SYSTEM TRAFFIC_LIGHT_CENTRALIZED (* System Configuration *)
  (* Standard: 61499-1 *)
  (* Version 0.4, 2009-03-05, JHC, Holobloc Inc., Deleted Application. *)
  (* Version 0.3, 2003-12-05, JHC, Rockwell Automation, Renamed from NEWSYSTEM. *)
  (* Version 0.2, 2002-11-05, JHC, Rockwell Automation, Fixed missing (empty) FBD in Application. *)
  (* Version 0.1, 2002-01-17, JHC, Rockwell Automation, Minor cleanup *)
  (* Version 0.0, 2000-05-27, JHC, Rockwell Automation *)
  DEVICE HMI_ROAD3_ROAD4 : FRAME_DEVICE(GRID := [2,1], BOUNDS := [10,10,300,500])
    RESOURCE HMI_ROAD3 : PANEL_RESOURCE
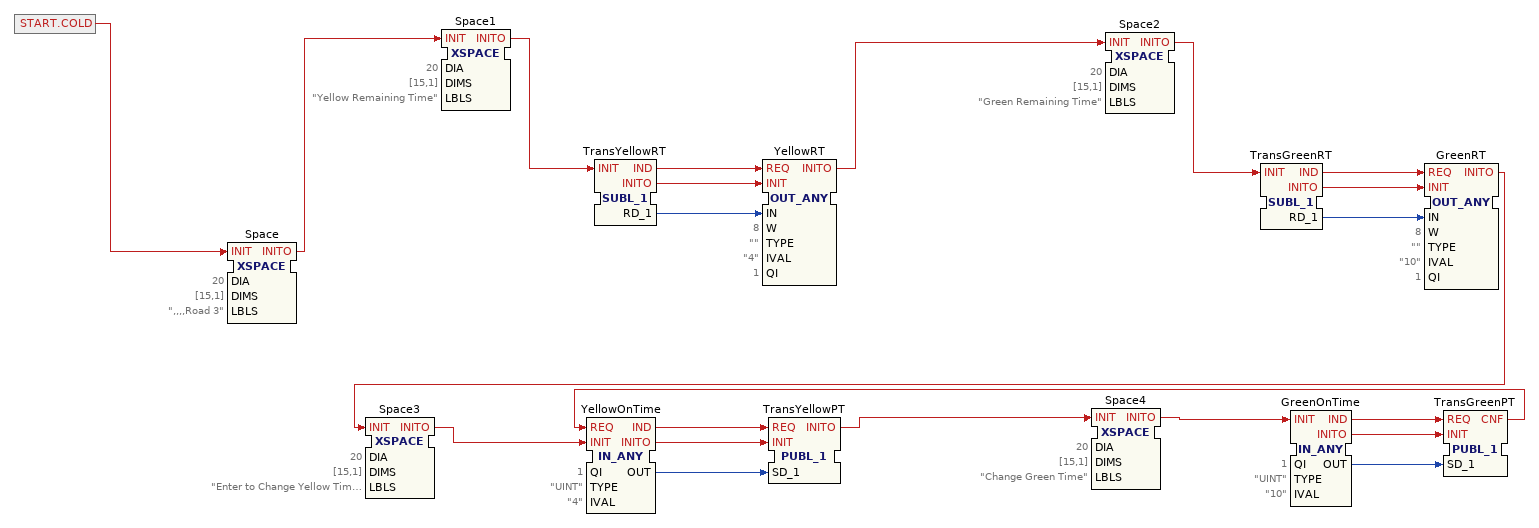
      FBS
        YellowRT : OUT_ANY(W := 8, TYPE := "", IVAL := "4", QI := 1);
        GreenRT : OUT_ANY(W := 8, TYPE := "", IVAL := "10", QI := 1);
        TransYellowRT : SUBL_1;
        TransGreenRT : SUBL_1;
        TransGreenPT : PUBL_1;
        TransYellowPT : PUBL_1;
        GreenOnTime : IN_ANY(QI := 1, TYPE := "UINT", IVAL := "10");
        YellowOnTime : IN_ANY(QI := 1, TYPE := "UINT", IVAL := "4");
        Space2 : XSPACE(DIA := 20, DIMS := [15,1], LBLS := "Green Remaining Time");
        Space1 : XSPACE(DIA := 20, DIMS := [15,1], LBLS := "Yellow Remaining Time");
        Space3 : XSPACE(DIA := 20, DIMS := [15,1], LBLS := "Enter to Change  Yellow Time");
        Space4 : XSPACE(DIA := 20, DIMS := [15,1], LBLS := "Change  Green Time");
        Space : XSPACE(DIA := 20, DIMS := [15,1], LBLS := ",,,,Road 3");
      END_FBS
      EVENT_CONNECTIONS
        TransYellowRT.IND TO YellowRT.REQ;
        TransGreenRT.IND TO GreenRT.REQ;
        YellowOnTime.IND TO TransYellowPT.REQ;
        GreenOnTime.IND TO TransGreenPT.REQ;
        YellowOnTime.INITO TO TransYellowPT.INIT;
        GreenOnTime.INITO TO TransGreenPT.INIT;
        TransGreenPT.CNF TO YellowOnTime.REQ;
        TransGreenRT.INITO TO GreenRT.INIT;
        YellowRT.INITO TO Space2.INIT;
        Space2.INITO TO TransGreenRT.INIT;
        TransYellowRT.INITO TO YellowRT.INIT;
        Space1.INITO TO TransYellowRT.INIT;
        GreenRT.INITO TO Space3.INIT;
        Space3.INITO TO YellowOnTime.INIT;
        TransYellowPT.INITO TO Space4.INIT;
        Space4.INITO TO GreenOnTime.INIT;
        START.COLD TO Space.INIT;
        Space.INITO TO Space1.INIT;
      END_CONNECTIONS
      DATA_CONNECTIONS
        TransYellowRT.RD_1 TO YellowRT.IN;
        TransGreenRT.RD_1 TO GreenRT.IN;
        YellowOnTime.OUT TO TransYellowPT.SD_1;
        GreenOnTime.OUT TO TransGreenPT.SD_1;
      END_CONNECTIONS
    END_RESOURCE
    RESOURCE HMI_ROAD4 : PANEL_RESOURCE
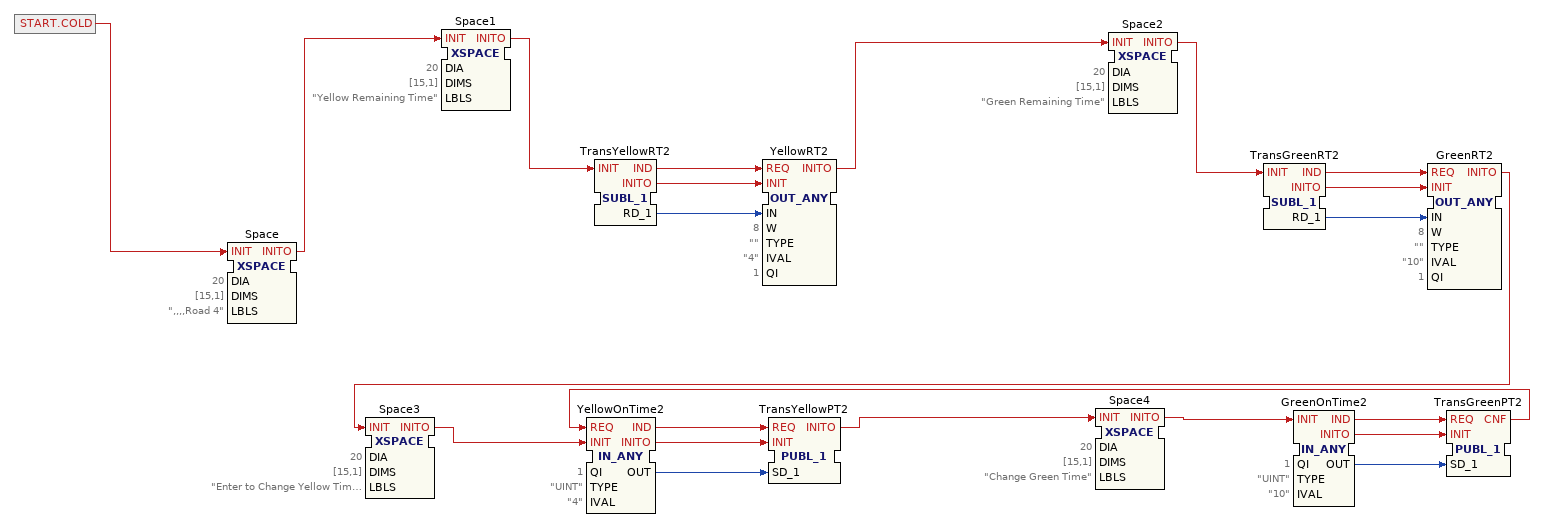
      FBS
        YellowRT2 : OUT_ANY(W := 8, TYPE := "", IVAL := "4", QI := 1);
        GreenRT2 : OUT_ANY(W := 8, TYPE := "", IVAL := "10", QI := 1);
        TransYellowRT2 : SUBL_1;
        TransGreenRT2 : SUBL_1;
        TransGreenPT2 : PUBL_1;
        TransYellowPT2 : PUBL_1;
        GreenOnTime2 : IN_ANY(QI := 1, TYPE := "UINT", IVAL := "10");
        YellowOnTime2 : IN_ANY(QI := 1, TYPE := "UINT", IVAL := "4");
        Space2 : XSPACE(DIA := 20, DIMS := [15,1], LBLS := "Green Remaining Time");
        Space1 : XSPACE(DIA := 20, DIMS := [15,1], LBLS := "Yellow Remaining Time");
        Space3 : XSPACE(DIA := 20, DIMS := [15,1], LBLS := "Enter to Change  Yellow Time");
        Space4 : XSPACE(DIA := 20, DIMS := [15,1], LBLS := "Change  Green Time");
        Space : XSPACE(DIA := 20, DIMS := [15,1], LBLS := ",,,,Road 4");
      END_FBS
      EVENT_CONNECTIONS
        TransYellowRT2.IND TO YellowRT2.REQ;
        TransGreenRT2.IND TO GreenRT2.REQ;
        YellowOnTime2.IND TO TransYellowPT2.REQ;
        GreenOnTime2.IND TO TransGreenPT2.REQ;
        YellowOnTime2.INITO TO TransYellowPT2.INIT;
        GreenOnTime2.INITO TO TransGreenPT2.INIT;
        TransGreenPT2.CNF TO YellowOnTime2.REQ;
        TransGreenRT2.INITO TO GreenRT2.INIT;
        YellowRT2.INITO TO Space2.INIT;
        Space2.INITO TO TransGreenRT2.INIT;
        TransYellowRT2.INITO TO YellowRT2.INIT;
        Space1.INITO TO TransYellowRT2.INIT;
        GreenRT2.INITO TO Space3.INIT;
        Space3.INITO TO YellowOnTime2.INIT;
        TransYellowPT2.INITO TO Space4.INIT;
        Space4.INITO TO GreenOnTime2.INIT;
        START.COLD TO Space.INIT;
        Space.INITO TO Space1.INIT;
      END_CONNECTIONS
      DATA_CONNECTIONS
        TransYellowRT2.RD_1 TO YellowRT2.IN;
        TransGreenRT2.RD_1 TO GreenRT2.IN;
        YellowOnTime2.OUT TO TransYellowPT2.SD_1;
        GreenOnTime2.OUT TO TransGreenPT2.SD_1;
      END_CONNECTIONS
    END_RESOURCE
  END_DEVICE
  DEVICE VIEW_ROAD3_ROAD4 : FRAME_DEVICE(BOUNDS := [310,10,300,500], GRID := [2,1])
    RESOURCE VIEW_ROAD3 : PANEL_RESOURCE(ROWS := 0, COLS := 0)
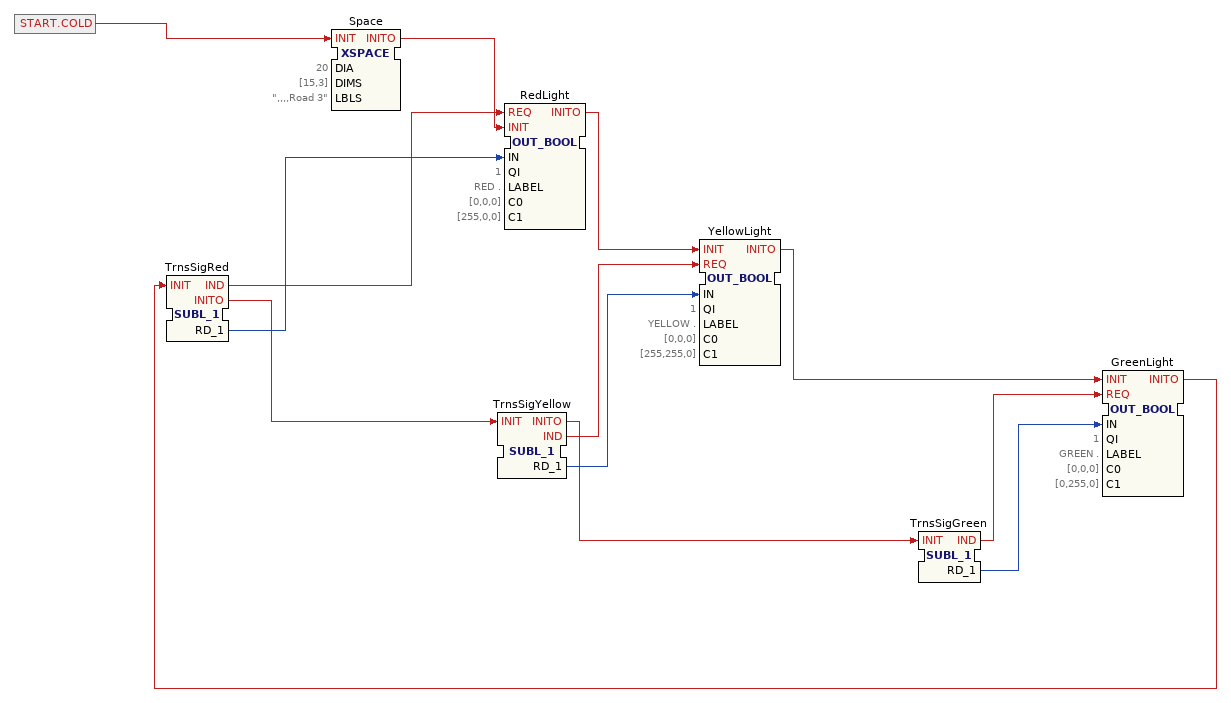
      FBS
        TrnsSigRed : SUBL_1;
        YellowLight : OUT_BOOL(QI := 1, LABEL := YELLOW    ., C0 := [0,0,0], C1 := [255,255,0]);
        RedLight : OUT_BOOL(QI := 1, LABEL := RED    ., C0 := [0,0,0], C1 := [255,0,0]);
        GreenLight : OUT_BOOL(QI := 1, LABEL := GREEN    ., C0 := [0,0,0], C1 := [0,255,0]);
        TrnsSigYellow : SUBL_1;
        TrnsSigGreen : SUBL_1;
        Space : XSPACE(DIA := 20, DIMS := [15,3], LBLS := ",,,,Road 3");
      END_FBS
      EVENT_CONNECTIONS
        RedLight.INITO TO YellowLight.INIT;
        YellowLight.INITO TO GreenLight.INIT;
        GreenLight.INITO TO TrnsSigRed.INIT;
        TrnsSigRed.IND TO RedLight.REQ;
        TrnsSigRed.INITO TO TrnsSigYellow.INIT;
        TrnsSigYellow.INITO TO TrnsSigGreen.INIT;
        TrnsSigYellow.IND TO YellowLight.REQ;
        TrnsSigGreen.IND TO GreenLight.REQ;
        START.COLD TO Space.INIT;
        Space.INITO TO RedLight.INIT;
      END_CONNECTIONS
      DATA_CONNECTIONS
        TrnsSigRed.RD_1 TO RedLight.IN;
        TrnsSigYellow.RD_1 TO YellowLight.IN;
        TrnsSigGreen.RD_1 TO GreenLight.IN;
      END_CONNECTIONS
    END_RESOURCE
    RESOURCE VIEW_ROAD4 : PANEL_RESOURCE(ROWS := 0, COLS := 0)
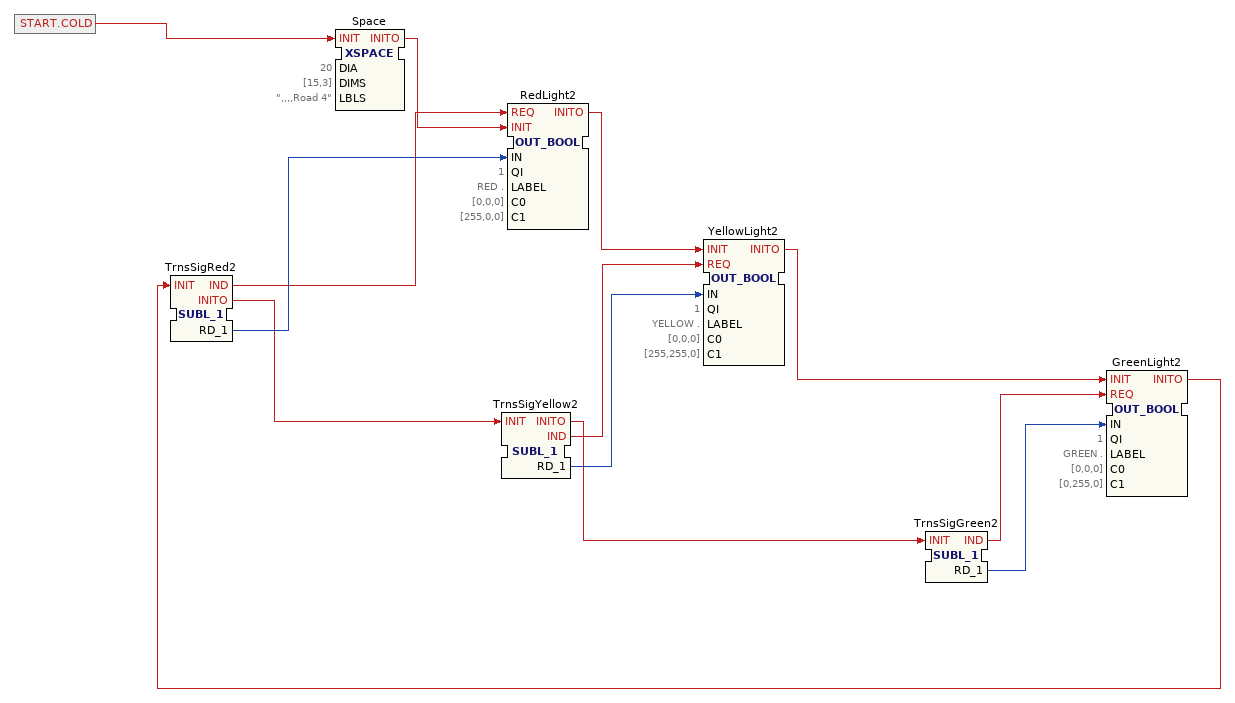
      FBS
        TrnsSigRed2 : SUBL_1;
        YellowLight2 : OUT_BOOL(QI := 1, LABEL := YELLOW    ., C0 := [0,0,0], C1 := [255,255,0]);
        RedLight2 : OUT_BOOL(QI := 1, LABEL := RED    ., C0 := [0,0,0], C1 := [255,0,0]);
        GreenLight2 : OUT_BOOL(QI := 1, LABEL := GREEN    ., C0 := [0,0,0], C1 := [0,255,0]);
        TrnsSigYellow2 : SUBL_1;
        TrnsSigGreen2 : SUBL_1;
        Space : XSPACE(DIA := 20, DIMS := [15,3], LBLS := ",,,,Road 4");
      END_FBS
      EVENT_CONNECTIONS
        RedLight2.INITO TO YellowLight2.INIT;
        YellowLight2.INITO TO GreenLight2.INIT;
        GreenLight2.INITO TO TrnsSigRed2.INIT;
        TrnsSigRed2.IND TO RedLight2.REQ;
        TrnsSigRed2.INITO TO TrnsSigYellow2.INIT;
        TrnsSigYellow2.INITO TO TrnsSigGreen2.INIT;
        TrnsSigYellow2.IND TO YellowLight2.REQ;
        TrnsSigGreen2.IND TO GreenLight2.REQ;
        START.COLD TO Space.INIT;
        Space.INITO TO RedLight2.INIT;
      END_CONNECTIONS
      DATA_CONNECTIONS
        TrnsSigRed2.RD_1 TO RedLight2.IN;
        TrnsSigYellow2.RD_1 TO YellowLight2.IN;
        TrnsSigGreen2.RD_1 TO GreenLight2.IN;
      END_CONNECTIONS
    END_RESOURCE
  END_DEVICE
  DEVICE MODEL_ROAD3_ROAD4 : FRAME_DEVICE(BOUNDS := [0,0,0,0], GRID := [1,1])
    RESOURCE MODEL_ROAD3 : PANEL_RESOURCE(ROWS := 0, COLS := 0)
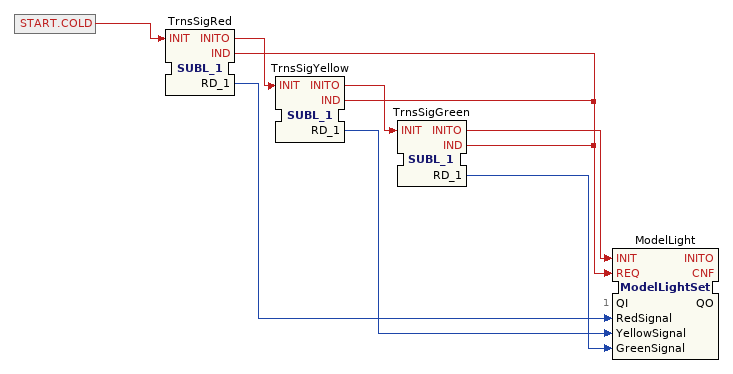
      FBS
        TrnsSigRed : SUBL_1;
        TrnsSigYellow : SUBL_1;
        TrnsSigGreen : SUBL_1;
        ModelLight : ModelLightSet(QI := 1);
      END_FBS
      EVENT_CONNECTIONS
        TrnsSigRed.INITO TO TrnsSigYellow.INIT;
        TrnsSigYellow.INITO TO TrnsSigGreen.INIT;
        START.COLD TO TrnsSigRed.INIT;
        TrnsSigGreen.INITO TO ModelLight.INIT;
        TrnsSigGreen.IND TO ModelLight.REQ;
        TrnsSigYellow.IND TO ModelLight.REQ;
        TrnsSigRed.IND TO ModelLight.REQ;
      END_CONNECTIONS
      DATA_CONNECTIONS
        TrnsSigRed.RD_1 TO ModelLight.RedSignal;
        TrnsSigYellow.RD_1 TO ModelLight.YellowSignal;
        TrnsSigGreen.RD_1 TO ModelLight.GreenSignal;
      END_CONNECTIONS
    END_RESOURCE
    RESOURCE MODEL_ROAD4 : PANEL_RESOURCE(ROWS := 0, COLS := 0)
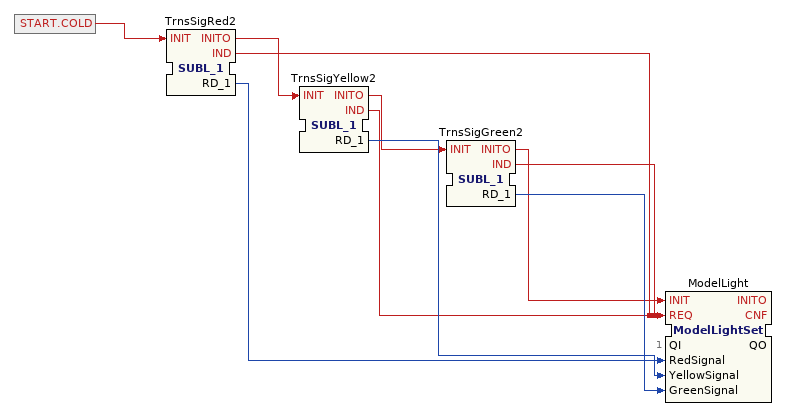
      FBS
        TrnsSigRed2 : SUBL_1;
        TrnsSigYellow2 : SUBL_1;
        TrnsSigGreen2 : SUBL_1;
        ModelLight : ModelLightSet(QI := 1);
      END_FBS
      EVENT_CONNECTIONS
        TrnsSigRed2.INITO TO TrnsSigYellow2.INIT;
        TrnsSigYellow2.INITO TO TrnsSigGreen2.INIT;
        START.COLD TO TrnsSigRed2.INIT;
        TrnsSigGreen2.INITO TO ModelLight.INIT;
        TrnsSigGreen2.IND TO ModelLight.REQ;
        TrnsSigYellow2.IND TO ModelLight.REQ;
        TrnsSigRed2.IND TO ModelLight.REQ;
      END_CONNECTIONS
      DATA_CONNECTIONS
        TrnsSigRed2.RD_1 TO ModelLight.RedSignal;
        TrnsSigYellow2.RD_1 TO ModelLight.YellowSignal;
        TrnsSigGreen2.RD_1 TO ModelLight.GreenSignal;
      END_CONNECTIONS
    END_RESOURCE
  END_DEVICE
  DEVICE CONTROL_ROAD3_ROAD4 : FRAME_DEVICE(BOUNDS := [0,0,0,0], GRID := [1,1])
    RESOURCE CENTRALIZE_CONTROL : PANEL_RESOURCE(ROWS := 0, COLS := 0)
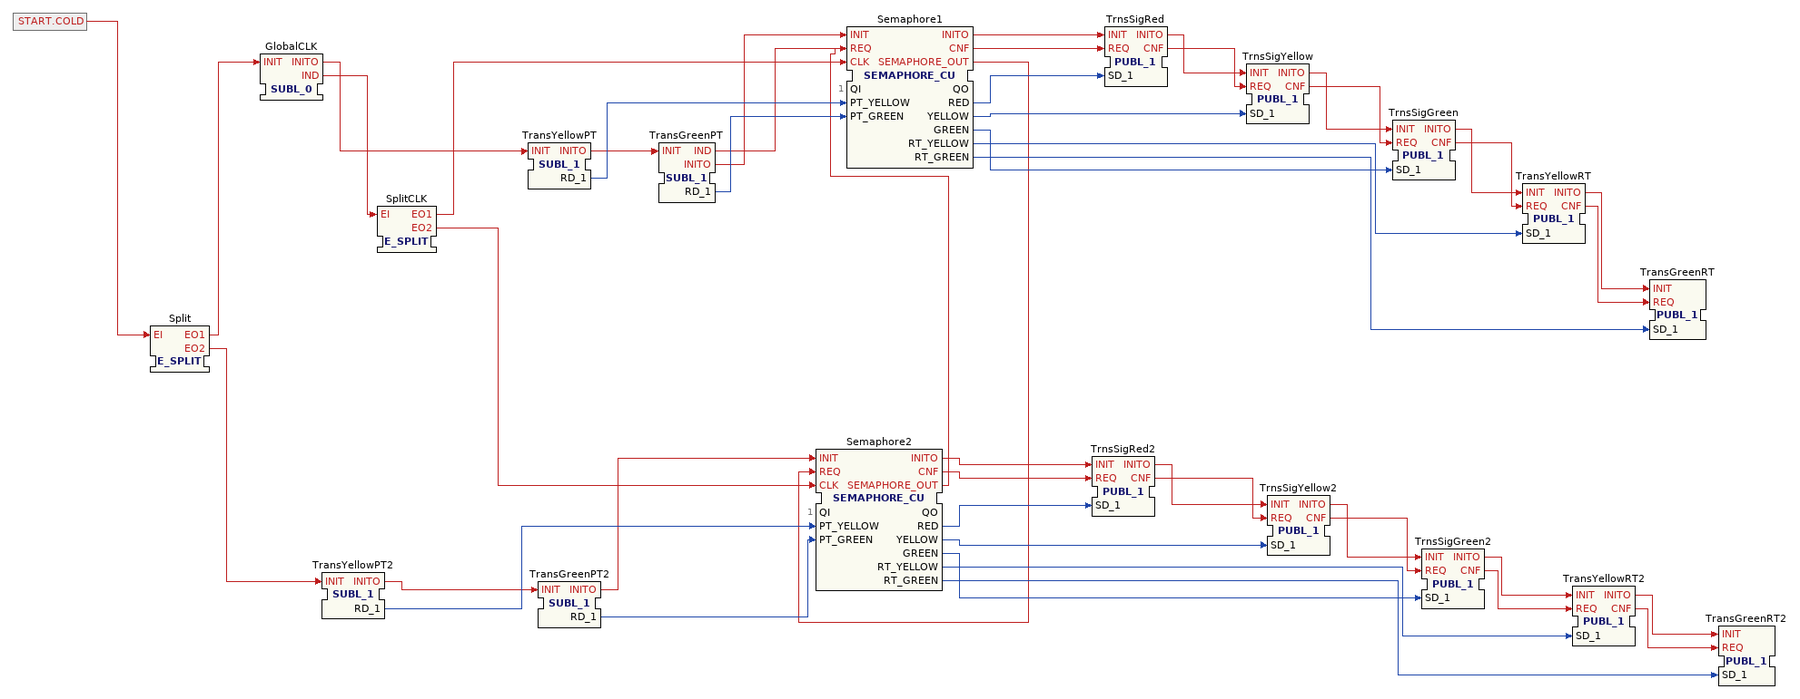
      FBS
        Semaphore1 : SEMAPHORE_CU(QI := 1);
        TrnsSigRed : PUBL_1;
        TrnsSigYellow : PUBL_1;
        TrnsSigGreen : PUBL_1;
        TransYellowRT : PUBL_1;
        TransGreenRT : PUBL_1;
        TransYellowPT : SUBL_1;
        TransGreenPT : SUBL_1;
        GlobalCLK : SUBL_0;
        TransYellowPT2 : SUBL_1;
        TransGreenPT2 : SUBL_1;
        Semaphore2 : SEMAPHORE_CU(QI := 1);
        TrnsSigRed2 : PUBL_1;
        TrnsSigYellow2 : PUBL_1;
        TrnsSigGreen2 : PUBL_1;
        TransYellowRT2 : PUBL_1;
        TransGreenRT2 : PUBL_1;
        Split : E_SPLIT;
        SplitCLK : E_SPLIT;
      END_FBS
      EVENT_CONNECTIONS
        Semaphore1.INITO TO TrnsSigRed.INIT;
        Semaphore1.CNF TO TrnsSigRed.REQ;
        TrnsSigRed.INITO TO TrnsSigYellow.INIT;
        TrnsSigRed.CNF TO TrnsSigYellow.REQ;
        TrnsSigYellow.INITO TO TrnsSigGreen.INIT;
        TrnsSigYellow.CNF TO TrnsSigGreen.REQ;
        TrnsSigGreen.INITO TO TransYellowRT.INIT;
        TrnsSigGreen.CNF TO TransYellowRT.REQ;
        TransYellowRT.INITO TO TransGreenRT.INIT;
        TransYellowRT.CNF TO TransGreenRT.REQ;
        TransYellowPT.INITO TO TransGreenPT.INIT;
        TransGreenPT.IND TO Semaphore1.REQ;
        GlobalCLK.INITO TO TransYellowPT.INIT;
        TransGreenPT.INITO TO Semaphore1.INIT;
        GlobalCLK.IND TO SplitCLK.EI;
        SplitCLK.EO1 TO Semaphore1.CLK;
        SplitCLK.EO2 TO Semaphore2.CLK;
        START.COLD TO Split.EI;
        Split.EO1 TO GlobalCLK.INIT;
        TransYellowPT2.INITO TO TransGreenPT2.INIT;
        Split.EO2 TO TransYellowPT2.INIT;
        TransGreenPT2.INITO TO Semaphore2.INIT;
        Semaphore2.INITO TO TrnsSigRed2.INIT;
        TrnsSigRed2.INITO TO TrnsSigYellow2.INIT;
        TrnsSigYellow2.INITO TO TrnsSigGreen2.INIT;
        TrnsSigGreen2.INITO TO TransYellowRT2.INIT;
        TransYellowRT2.INITO TO TransGreenRT2.INIT;
        TrnsSigRed2.CNF TO TrnsSigYellow2.REQ;
        TrnsSigYellow2.CNF TO TrnsSigGreen2.REQ;
        TrnsSigGreen2.CNF TO TransYellowRT2.REQ;
        TransYellowRT2.CNF TO TransGreenRT2.REQ;
        Semaphore2.CNF TO TrnsSigRed2.REQ;
        Semaphore1.SEMAPHORE_OUT TO Semaphore2.REQ;
        Semaphore2.SEMAPHORE_OUT TO Semaphore1.REQ;
      END_CONNECTIONS
      DATA_CONNECTIONS
        Semaphore1.RED TO TrnsSigRed.SD_1;
        Semaphore1.YELLOW TO TrnsSigYellow.SD_1;
        Semaphore1.GREEN TO TrnsSigGreen.SD_1;
        Semaphore1.RT_YELLOW TO TransYellowRT.SD_1;
        Semaphore1.RT_GREEN TO TransGreenRT.SD_1;
        TransYellowPT.RD_1 TO Semaphore1.PT_YELLOW;
        TransGreenPT.RD_1 TO Semaphore1.PT_GREEN;
        Semaphore2.RED TO TrnsSigRed2.SD_1;
        Semaphore2.YELLOW TO TrnsSigYellow2.SD_1;
        Semaphore2.GREEN TO TrnsSigGreen2.SD_1;
        Semaphore2.RT_YELLOW TO TransYellowRT2.SD_1;
        Semaphore2.RT_GREEN TO TransGreenRT2.SD_1;
        TransGreenPT2.RD_1 TO Semaphore2.PT_GREEN;
        TransYellowPT2.RD_1 TO Semaphore2.PT_YELLOW;
      END_CONNECTIONS
    END_RESOURCE
    RESOURCE GLOBAL_CLK : PANEL_RESOURCE
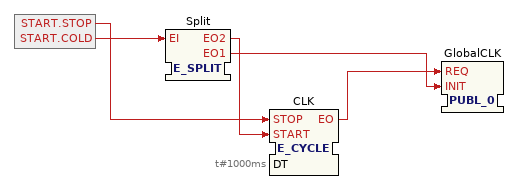
      FBS
        CLK : E_CYCLE(DT := t#1000ms);
        GlobalCLK : PUBL_0;
        Split : E_SPLIT;
      END_FBS
      EVENT_CONNECTIONS
        START.STOP TO CLK.STOP;
        CLK.EO TO GlobalCLK.REQ;
        START.COLD TO Split.EI;
        Split.EO2 TO CLK.START;
        Split.EO1 TO GlobalCLK.INIT;
      END_CONNECTIONS
    END_RESOURCE
  END_DEVICE
END_SYSTEM
